FUNCTION_BLOCK DRILL_SWITCH (* Drill event switcher *)
  (* Standard: 61499-2 *)
  (* Version 1.0, 11-01-12, GASR, Universidade do Estado de Santa Catarina *)
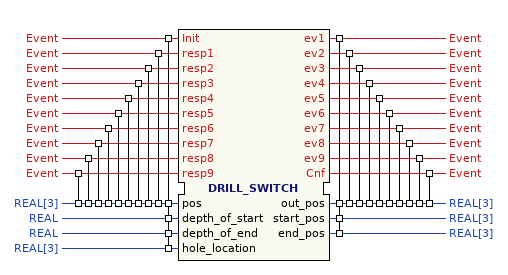
  EVENT_INPUT
    Init WITH pos, depth_of_start, depth_of_end, hole_location;
    resp1 WITH pos;
    resp2 WITH pos;
    resp3 WITH pos;
    resp4 WITH pos;
    resp5 WITH pos;
    resp6 WITH pos;
    resp7 WITH pos;
    resp8 WITH pos;
    resp9 WITH pos;
  END_EVENT
  EVENT_OUTPUT
    ev1 WITH out_pos, start_pos, end_pos;
    ev2 WITH out_pos;
    ev3 WITH out_pos;
    ev4 WITH out_pos;
    ev5 WITH out_pos;
    ev6 WITH out_pos;
    ev7 WITH out_pos;
    ev8 WITH out_pos;
    ev9 WITH out_pos;
    Cnf WITH out_pos;
  END_EVENT
  VAR_INPUT
    pos : ARRAY [0..2] OF REAL; (* Machine position *)
    depth_of_start : REAL := 0; (* Depth at which 'start' milling conditions are applyed *)
    depth_of_end : REAL := 0; (* Depth at which 'end' milling conditions are applyed *)
    hole_location : ARRAY [0..2] OF REAL; (* Feature location coordinates *)
  END_VAR
  VAR_OUTPUT
    out_pos : ARRAY [0..2] OF REAL; (* Machine position *)
    start_pos : ARRAY [0..2] OF REAL; (* Position at which 'start' milling conditions are applyed *)
    end_pos : ARRAY [0..2] OF REAL; (* Position at which 'end' milling conditions are applyed *)
  END_VAR
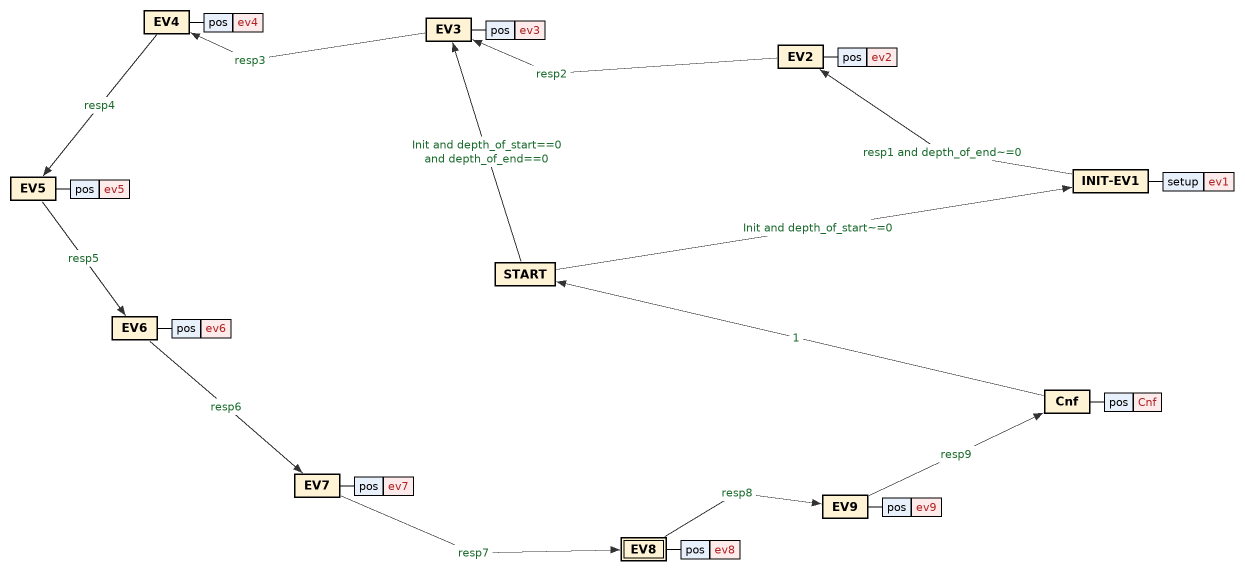
  EC_STATES
    EV8 : pos -> ev8;
    EV4 : pos -> ev4;
    EV3 : pos -> ev3;
    EV6 : pos -> ev6;
    EV9 : pos -> ev9;
    Cnf : pos -> Cnf;
    INIT-EV1 : setup -> ev1;
    EV2 : pos -> ev2;
    EV5 : pos -> ev5;
    START;
    EV7 : pos -> ev7;
  END_STATES
  EC_TRANSITIONS
    START TO INIT-EV1 := Init and depth_of_start~=0;
    INIT-EV1 TO EV2 := resp1 and depth_of_end~=0;
    START TO EV3 := Init and depth_of_start==0 and depth_of_end==0;
    EV2 TO EV3 := resp2;
    EV3 TO EV4 := resp3;
    EV4 TO EV5 := resp4;
    EV5 TO EV6 := resp5;
    EV6 TO EV7 := resp6;
    EV7 TO EV8 := resp7;
    EV8 TO EV9 := resp8;
    EV9 TO Cnf := resp9;
    Cnf TO START := 1;
  END_TRANSITIONS
  ALGORITHM pos IN Lua:
 print( pos[1], pos[2], pos[3] ) out_pos[ 1 ] = pos[ 1 ] out_pos[ 2 ] = pos[ 2 ] out_pos[ 3 ] = pos[ 3 ]
  END_ALGORITHM
  ALGORITHM setup IN Lua:
 print( pos[1], pos[2], pos[3], 'depths', depth_of_start, depth_of_end ) out_pos[ 1 ] = pos[ 1 ] out_pos[ 2 ] = pos[ 2 ] out_pos[ 3 ] = pos[ 3 ] start_pos[ 1 ] = hole_location[ 1 ] start_pos[ 2 ] = hole_location[ 2 ] start_pos[ 3 ] = hole_location[ 3 ] start_pos[ 3 ] = hole_location[ 3 ] - depth_of_start end_pos[ 1 ] = hole_location[ 1 ] end_pos[ 2 ] = hole_location[ 2 ] end_pos[ 3 ] = hole_location[ 3 ] end_pos[ 3 ] = hole_location[ 3 ] - depth_of_end
  END_ALGORITHM
END_FUNCTION_BLOCK
